// TIA Portal V21 export
FUNCTION "PassiLavaggio_010102" : Void   // FC102, LAD
{ S7_Optimized_Access := 'TRUE' }
// stored: SetENOAutomatically false
   VAR_TEMP
      CondizioniPassoEsterne : Bool;
      AbilitazionePasso : Bool;
      AppoggioComando : Int;
      ComandoValvolaG : Int;
      ComandoValvolaA1 : Int;
      PompaPistoniAbilitata : Bool;
   END_VAR
   VAR CONSTANT
      Positivo : Int := 2;
      Negativo : Int := 3;
      FolleScarico : Int := 4;
      FlipFlop : Int := 5;
   END_VAR
BEGIN

REGION Network 1: Sequenza: Lavaggio - Passo: Risciacquo. Condizioni passo esterne.
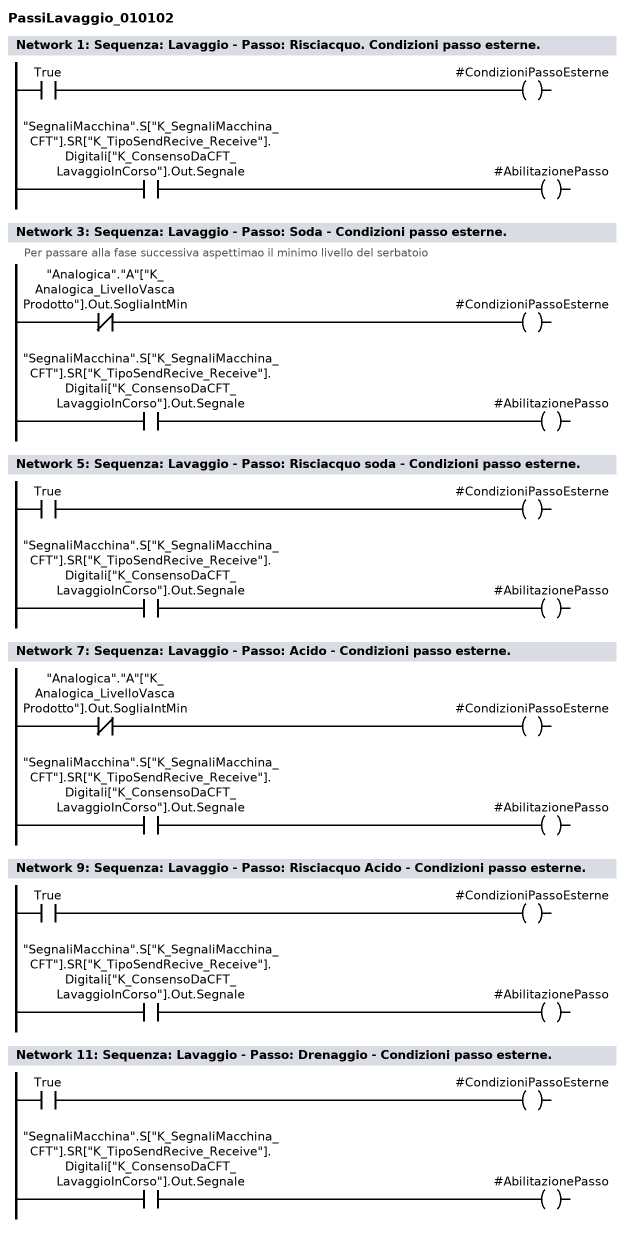
   RUNG wire#powerrail
      Contact( True )
      Coil( #CondizioniPassoEsterne )
   END_RUNG
   RUNG wire#powerrail
      Contact( "SegnaliMacchina".S["K_SegnaliMacchina_CFT"].SR["K_TipoSendRecive_Receive"].Digitali["K_ConsensoDaCFT_LavaggioInCorso"].Out.Segnale )
      Coil( #AbilitazionePasso )
   END_RUNG
   // the same network as SCL:
   #CondizioniPassoEsterne := True;
   #AbilitazionePasso := "SegnaliMacchina".S["K_SegnaliMacchina_CFT"].SR["K_TipoSendRecive_Receive"].Digitali["K_ConsensoDaCFT_LavaggioInCorso"].Out.Segnale;
END_REGION

REGION Network 2 (SCL): Sequenza: Lavaggio - Passo: Risciacquo. Gestione del passo.
   REGION Parametri del passo
       "GestPasso"(K_PassoAttuale := "K_Passo_Risciacquo",
                   K_PassoSuccessivo := "K_Passo_Soda",
                   AbilitaSaltapasso := True,
                   AbilitaPasso:= #AbilitazionePasso,
                   CondizioniPassoEsterne := #CondizioniPassoEsterne,
                   K_Sequenza := "K_Sequenza_Lavaggio");
   END_REGION ;
   REGION Comando delle utenze nel passo

       "GestPasso_CmdValvola"(K_Valvola := "K_Valvola_A1",
                              Comando := #Positivo,
                              K_Sequenza := "K_Sequenza_Lavaggio",
                              K_Passo := "K_Passo_Risciacquo",
                              NonAttenderePosizione:= "Analogica".A[K_Analogica_LivelloVascaProdotto].Out.SogliaIntMax);

       "GestPasso_CmdValvola"(K_Valvola := "K_Valvola_A",
                              Comando := #Positivo,
                              K_Sequenza := "K_Sequenza_Lavaggio",
                              K_Passo := "K_Passo_Risciacquo",
                              NonAttenderePosizione := "Analogica".A[K_Analogica_LivelloVascaProdotto].Out.SogliaIntMax);

       "GestPasso_CmdValvolaFlipFlop"(K_Valvola := "K_Valvola_B",
                                      NumeroCicli := 3,
                                      TempoPositivo := "Sequenza".S[K_Sequenza_Lavaggio].Prm.Passo[K_Passo_Risciacquo].Durata.Preset / 3,  //Tempo a ricetta per immissione soda
                                      TempoNegativo := 5,
                                      ComandoARiposo:=#Positivo,
                                      K_Sequenza := "K_Sequenza_Lavaggio",
                                      K_Passo := "K_Passo_Risciacquo");

       "GestPasso_CmdValvola"(K_Valvola := "K_Valvola_B1",
                              Comando := "GestPasso_ReplicaComandoValvola"("K_Valvola_B"),
                              K_Sequenza := "K_Sequenza_Lavaggio",
                              K_Passo := "K_Passo_Risciacquo",
                              NonAttenderePosizione:= False);

       "GestPasso_CmdValvola"(K_Valvola := "K_Valvola_E",
                              Comando := #Positivo,
                              K_Sequenza := "K_Sequenza_Lavaggio",
                              K_Passo := "K_Passo_Risciacquo",
                              NonAttenderePosizione:= False);

       "GestPasso_CmdValvola"(K_Valvola := "K_Valvola_E1",
                              Comando := #Positivo,
                              K_Sequenza := "K_Sequenza_Lavaggio",
                              K_Passo := "K_Passo_Risciacquo",
                              NonAttenderePosizione:= False);

       "GestPasso_CmdValvola"(K_Valvola := "K_Valvola_G",
                              Comando := #Positivo,
                              K_Sequenza := "K_Sequenza_Lavaggio",
                              K_Passo := "K_Passo_Risciacquo",
                              NonAttenderePosizione := False);

       "GestPasso_CmdValvolaFlipFlop"(K_Valvola := "K_Valvola_CP1",
                                      NumeroCicli := 5,
                                      TempoPositivo := "Sequenza".S[K_Sequenza_Lavaggio].Prm.Passo[K_Passo_Risciacquo].Durata.Preset / 5,
                                      TempoNegativo := 5,
                                      ComandoARiposo:=#Positivo,
                                      K_Passo := "K_Passo_Risciacquo",
                                      K_Sequenza := "K_Sequenza_Lavaggio");

       "GestPasso_CmdMotore"(K_Motore := "K_Motore_PompaMono",
                             Comando := #Positivo,
                             K_Sequenza := "K_Sequenza_Lavaggio",
                             K_Passo := "K_Passo_Risciacquo",
                             NonAttenderePosizione := False);
       #PompaPistoniAbilitata := "MacchinaARicetta".M[K_MacchinaARicetta_SterilizzatoreTubo].Lavoro.DatoBool[K_DatoRicettaBool_SterilizzatoreTubo_AbilitazionePompaPistoni];
       IF #PompaPistoniAbilitata THEN
           "GestPasso_CmdMotore"(K_Motore := "K_Motore_PompaPistoni",
                                 Comando := #Positivo,
                                 K_Sequenza := "K_Sequenza_Lavaggio",
                                 K_Passo := "K_Passo_Risciacquo",
                                 NonAttenderePosizione := NOT "MacchinaARicetta".M[K_MacchinaARicetta_SterilizzatoreTubo].Lavoro.DatoBool[K_DatoRicettaBool_SterilizzatoreTubo_AbilitazionePompaPistoni]);
       END_IF;
       "GestPasso_CmdMotore"(K_Motore := "K_Motore_CentrifugaLavaggio",
                             Comando := #Positivo,
                             K_Sequenza := "K_Sequenza_Lavaggio",
                             K_Passo := "K_Passo_Risciacquo",
                             NonAttenderePosizione := False);
   END_REGION ;
END_REGION

REGION Network 3: Sequenza: Lavaggio - Passo: Soda - Condizioni passo esterne.
   // Per passare alla fase successiva aspettimao il minimo livello del serbatoio
   RUNG wire#powerrail
      I_Contact( "Analogica"."A"["K_Analogica_LivelloVascaProdotto"].Out.SogliaIntMin )
      Coil( #CondizioniPassoEsterne )
   END_RUNG
   RUNG wire#powerrail
      Contact( "SegnaliMacchina".S["K_SegnaliMacchina_CFT"].SR["K_TipoSendRecive_Receive"].Digitali["K_ConsensoDaCFT_LavaggioInCorso"].Out.Segnale )
      Coil( #AbilitazionePasso )
   END_RUNG
   // the same network as SCL:
   #CondizioniPassoEsterne := NOT "Analogica"."A"["K_Analogica_LivelloVascaProdotto"].Out.SogliaIntMin;
   #AbilitazionePasso := "SegnaliMacchina".S["K_SegnaliMacchina_CFT"].SR["K_TipoSendRecive_Receive"].Digitali["K_ConsensoDaCFT_LavaggioInCorso"].Out.Segnale;
END_REGION

REGION Network 4 (SCL): Sequenza: Lavaggio - Passo: Soda - Gestione del passo.
   REGION Parametri del passo
       "GestPasso"(K_PassoAttuale := "K_Passo_Soda",
                   K_PassoSuccessivo := "K_Passo_RisciacquoSoda",
                   AbilitaSaltapasso := True,
                   AbilitaPasso:= #AbilitazionePasso,
                   CondizioniPassoEsterne := #CondizioniPassoEsterne,
                   K_Sequenza := "K_Sequenza_Lavaggio");
   END_REGION ;
   REGION Comando delle utenze nel passo    
       IF "Sequenza".S[K_Sequenza_Lavaggio].Prm.Passo[K_Passo_Soda].Durata.O THEN
           #ComandoValvolaA1 := #Negativo;
       ELSE
           #ComandoValvolaA1 := #Positivo;
       END_IF;
       "GestPasso_CmdValvola"(K_Valvola := "K_Valvola_A1",
                              Comando := #ComandoValvolaA1,
                              K_Sequenza := "K_Sequenza_Lavaggio",
                              K_Passo := "K_Passo_Soda",
                              NonAttenderePosizione:= "Analogica".A[K_Analogica_LivelloVascaProdotto].Out.SogliaIntMax);

       "GestPasso_CmdValvola"(K_Valvola := "K_Valvola_A",
                              Comando := #ComandoValvolaA1,
                              K_Sequenza := "K_Sequenza_Lavaggio",
                              K_Passo := "K_Passo_Soda",
                              NonAttenderePosizione := "Analogica".A[K_Analogica_LivelloVascaProdotto].Out.SogliaIntMax);

       "GestPasso_CmdValvolaFlipFlop"(K_Valvola := "K_Valvola_B",
                                      NumeroCicli := 8,
                                      TempoPositivo := "Sequenza".S[K_Sequenza_Lavaggio].Prm.Passo[K_Passo_Soda].Durata.Preset / 8,
                                      TempoNegativo := 5,
                                      ComandoARiposo:=#Positivo,
                                      K_Passo := "K_Passo_Soda",
                                      K_Sequenza := "K_Sequenza_Lavaggio");

       "GestPasso_CmdValvola"(K_Valvola := "K_Valvola_B1",
                              Comando := "GestPasso_ReplicaComandoValvola"("K_Valvola_B"),
                              K_Sequenza := "K_Sequenza_Lavaggio",
                              K_Passo := "K_Passo_Soda",
                              NonAttenderePosizione:= False);

       "GestPasso_CmdValvola"(K_Valvola := "K_Valvola_D",
                              Comando := #Positivo,
                              K_Sequenza := "K_Sequenza_Lavaggio",
                              K_Passo := "K_Passo_Soda",
                              NonAttenderePosizione:= False);

       "GestPasso_CmdValvola"(K_Valvola := "K_Valvola_D2",
                              Comando :=#Positivo,
                              K_Sequenza := "K_Sequenza_Lavaggio",
                              K_Passo := "K_Passo_Soda",
                              NonAttenderePosizione:= False);

       "GestPasso_CmdValvola"(K_Valvola := "K_Valvola_E",
                              Comando := #Positivo,
                              K_Sequenza := "K_Sequenza_Lavaggio",
                              K_Passo := "K_Passo_Soda",
                              NonAttenderePosizione:= False);

       "GestPasso_CmdValvola"(K_Valvola := "K_Valvola_E1",
                              Comando := #Positivo,
                              K_Sequenza := "K_Sequenza_Lavaggio",
                              K_Passo := "K_Passo_Soda",
                              NonAttenderePosizione:= False);

       REGION Valvola G
           //Al termine del passo prima di passare al passo successivo aspetto il livello minimo,
           //quindi metto in scarico invece di andare in vasca.
           IF "Sequenza".S[K_Sequenza_Lavaggio].Prm.Passo[K_Passo_Soda].Durata.O THEN
               #ComandoValvolaG := #Positivo;
           ELSE
               #ComandoValvolaG := #Negativo;
           END_IF;

           "GestPasso_CmdValvola"(K_Valvola := "K_Valvola_G",
                                  Comando := #ComandoValvolaG,
                                  K_Sequenza := "K_Sequenza_Lavaggio",
                                  K_Passo := "K_Passo_Soda",
                                  NonAttenderePosizione := False);
       END_REGION ;

       "GestPasso_CmdValvola"(K_Valvola := "K_Valvola_Z1",
                              Comando := "GestPasso_ReplicaComandoValvola"("K_Valvola_XXX"),
                              K_Sequenza := "K_Sequenza_Lavaggio",
                              K_Passo := "K_Passo_Soda",
                              NonAttenderePosizione:= False);

       "GestPasso_CmdValvolaFlipFlop"(K_Valvola := "K_Valvola_XXX",
                                      NumeroCicli := 1,
                                      TempoPositivo := 300,  //Tempo per immissione soda
                                      TempoNegativo := 0,
                                      ComandoARiposo:=#Negativo,
                                      K_Sequenza := "K_Sequenza_Lavaggio",
                                      K_Passo := "K_Passo_Soda");

       "GestPasso_CmdValvolaFlipFlop"(K_Valvola := "K_Valvola_CP1",
                                      NumeroCicli := 5,
                                      TempoPositivo := "Sequenza".S[K_Sequenza_Lavaggio].Prm.Passo[K_Passo_Soda].Durata.Preset / 5,
                                      TempoNegativo := 5,
                                      ComandoARiposo:=#Positivo,
                                      K_Passo := "K_Passo_Soda",
                                      K_Sequenza := "K_Sequenza_Lavaggio");
       //Motori
       "GestPasso_CmdMotore"(K_Motore := "K_Motore_PompaMono",
                             Comando := #Positivo,
                             K_Sequenza := "K_Sequenza_Lavaggio",
                             K_Passo := "K_Passo_Soda",
                             NonAttenderePosizione := False);
       IF #PompaPistoniAbilitata THEN
           "GestPasso_CmdMotore"(K_Motore := "K_Motore_PompaPistoni",
                                 Comando := #Positivo,
                                 K_Sequenza := "K_Sequenza_Lavaggio",
                                 K_Passo := "K_Passo_Soda",
                                 NonAttenderePosizione := NOT "MacchinaARicetta".M[K_MacchinaARicetta_SterilizzatoreTubo].Lavoro.DatoBool[K_DatoRicettaBool_SterilizzatoreTubo_AbilitazionePompaPistoni]);
       END_IF;
       "GestPasso_CmdMotore"(K_Motore := "K_Motore_CentrifugaLavaggio",
                             Comando := #Positivo,
                             K_Sequenza := "K_Sequenza_Lavaggio",
                             K_Passo := "K_Passo_Soda",
                             NonAttenderePosizione := False);

       "GestPasso_CmdMotore"(K_Motore := "K_Motore_PompaRicircoloAcquaCalda",
                             Comando := #Positivo,
                             K_Sequenza := "K_Sequenza_Lavaggio",
                             K_Passo := "K_Passo_Soda",
                             NonAttenderePosizione := False);

   END_REGION ;
END_REGION

REGION Network 5: Sequenza: Lavaggio - Passo: Risciacquo soda - Condizioni passo esterne.
   RUNG wire#powerrail
      Contact( True )
      Coil( #CondizioniPassoEsterne )
   END_RUNG
   RUNG wire#powerrail
      Contact( "SegnaliMacchina".S["K_SegnaliMacchina_CFT"].SR["K_TipoSendRecive_Receive"].Digitali["K_ConsensoDaCFT_LavaggioInCorso"].Out.Segnale )
      Coil( #AbilitazionePasso )
   END_RUNG
   // the same network as SCL:
   #CondizioniPassoEsterne := True;
   #AbilitazionePasso := "SegnaliMacchina".S["K_SegnaliMacchina_CFT"].SR["K_TipoSendRecive_Receive"].Digitali["K_ConsensoDaCFT_LavaggioInCorso"].Out.Segnale;
END_REGION

REGION Network 6 (SCL): Sequenza: Lavaggio - Passo: Risciacquo soda - Gestione del passo.
   REGION Parametri del passo
   "GestPasso"(K_PassoAttuale := "K_Passo_RisciacquoSoda",
               K_PassoSuccessivo := "K_Passo_Acido",
               AbilitaSaltapasso := True,
               AbilitaPasso:= #AbilitazionePasso,
               CondizioniPassoEsterne := #CondizioniPassoEsterne,
               K_Sequenza := "K_Sequenza_Lavaggio");
   END_REGION ;
   REGION Comando delle utenze nel passo
       "GestPasso_CmdValvola"(K_Valvola := "K_Valvola_A1",
                              Comando := #Positivo,
                              K_Sequenza := "K_Sequenza_Lavaggio",
                              K_Passo := "K_Passo_RisciacquoSoda",
                              NonAttenderePosizione := "Analogica".A[K_Analogica_LivelloVascaProdotto].Out.SogliaIntMax);

       "GestPasso_CmdValvola"(K_Valvola := "K_Valvola_A",
                              Comando := #Positivo,
                              K_Sequenza := "K_Sequenza_Lavaggio",
                              K_Passo := "K_Passo_RisciacquoSoda",
                              NonAttenderePosizione := "Analogica".A[K_Analogica_LivelloVascaProdotto].Out.SogliaIntMax);

       "GestPasso_CmdValvolaFlipFlop"(K_Valvola := "K_Valvola_B",
                                      NumeroCicli := 3,
                                      TempoPositivo := "Sequenza".S[K_Sequenza_Lavaggio].Prm.Passo[K_Passo_RisciacquoSoda].Durata.Preset / 3,  //Tempo a ricetta per immissione soda
                                      TempoNegativo := 5,
                                      ComandoARiposo:=#Positivo,
                                      K_Sequenza := "K_Sequenza_Lavaggio",
                                      K_Passo := "K_Passo_RisciacquoSoda");

       "GestPasso_CmdValvola"(K_Valvola := "K_Valvola_B1",
                              Comando := "GestPasso_ReplicaComandoValvola"("K_Valvola_B"),
                              K_Sequenza := "K_Sequenza_Lavaggio",
                              K_Passo := "K_Passo_RisciacquoSoda",
                              NonAttenderePosizione := False);

       "GestPasso_CmdValvola"(K_Valvola := "K_Valvola_E",
                              Comando := #Positivo,
                              K_Sequenza := "K_Sequenza_Lavaggio",
                              K_Passo := "K_Passo_RisciacquoSoda",
                              NonAttenderePosizione := False);

       "GestPasso_CmdValvola"(K_Valvola := "K_Valvola_E1",
                              Comando := #Positivo,
                              K_Sequenza := "K_Sequenza_Lavaggio",
                              K_Passo := "K_Passo_RisciacquoSoda",
                              NonAttenderePosizione := False);

       "GestPasso_CmdValvola"(K_Valvola := "K_Valvola_G",
                              Comando := #Positivo,
                              K_Sequenza := "K_Sequenza_Lavaggio",
                              K_Passo := "K_Passo_RisciacquoSoda",
                              NonAttenderePosizione := False);

       "GestPasso_CmdValvolaFlipFlop"(K_Valvola := "K_Valvola_CP1",
                                      NumeroCicli := 5,
                                      TempoPositivo := "Sequenza".S[K_Sequenza_Lavaggio].Prm.Passo[K_Passo_RisciacquoSoda].Durata.Preset / 5,
                                      TempoNegativo := 5,
                                      ComandoARiposo:=#Positivo,
                                      K_Passo := "K_Passo_RisciacquoSoda",
                                      K_Sequenza := "K_Sequenza_Lavaggio");

       "GestPasso_CmdMotore"(K_Motore := "K_Motore_PompaMono",
                             Comando := #Positivo,
                             K_Sequenza := "K_Sequenza_Lavaggio",
                             K_Passo := "K_Passo_RisciacquoSoda",
                             NonAttenderePosizione := False);
       IF #PompaPistoniAbilitata THEN
           "GestPasso_CmdMotore"(K_Motore := "K_Motore_PompaPistoni",
                                 Comando := #Positivo,
                                 K_Sequenza := "K_Sequenza_Lavaggio",
                                 K_Passo := "K_Passo_RisciacquoSoda",
                                 NonAttenderePosizione := NOT "MacchinaARicetta".M[K_MacchinaARicetta_SterilizzatoreTubo].Lavoro.DatoBool[K_DatoRicettaBool_SterilizzatoreTubo_AbilitazionePompaPistoni]);
       END_IF;
       "GestPasso_CmdMotore"(K_Motore := "K_Motore_CentrifugaLavaggio",
                             Comando := #Positivo,
                             K_Sequenza := "K_Sequenza_Lavaggio",
                             K_Passo := "K_Passo_RisciacquoSoda",
                             NonAttenderePosizione := False);
   END_REGION ;
END_REGION

REGION Network 7: Sequenza: Lavaggio - Passo: Acido - Condizioni passo esterne.
   RUNG wire#powerrail
      I_Contact( "Analogica"."A"["K_Analogica_LivelloVascaProdotto"].Out.SogliaIntMin )
      Coil( #CondizioniPassoEsterne )
   END_RUNG
   RUNG wire#powerrail
      Contact( "SegnaliMacchina".S["K_SegnaliMacchina_CFT"].SR["K_TipoSendRecive_Receive"].Digitali["K_ConsensoDaCFT_LavaggioInCorso"].Out.Segnale )
      Coil( #AbilitazionePasso )
   END_RUNG
   // the same network as SCL:
   #CondizioniPassoEsterne := NOT "Analogica"."A"["K_Analogica_LivelloVascaProdotto"].Out.SogliaIntMin;
   #AbilitazionePasso := "SegnaliMacchina".S["K_SegnaliMacchina_CFT"].SR["K_TipoSendRecive_Receive"].Digitali["K_ConsensoDaCFT_LavaggioInCorso"].Out.Segnale;
END_REGION

REGION Network 8 (SCL): Sequenza: Lavaggio - Passo: Acido - Gestione del passo.
   REGION Parametri del passo
       "GestPasso"(K_PassoAttuale := "K_Passo_Acido",
                   K_PassoSuccessivo := "K_Passo_RisciacquoAcido",
                   AbilitaSaltapasso := True,
                   AbilitaPasso:= #AbilitazionePasso,
                   CondizioniPassoEsterne := #CondizioniPassoEsterne,
                   K_Sequenza := "K_Sequenza_Lavaggio");
   END_REGION ;
   REGION Comando delle utenze nel passo    
       IF "Sequenza".S[K_Sequenza_Lavaggio].Prm.Passo[K_Passo_Acido].Durata.O THEN
           #ComandoValvolaA1 := #Negativo;
       ELSE
           #ComandoValvolaA1 := #Positivo;
       END_IF;
       "GestPasso_CmdValvola"(K_Valvola := "K_Valvola_A1",
                              Comando := #ComandoValvolaA1,
                              K_Sequenza := "K_Sequenza_Lavaggio",
                              K_Passo := "K_Passo_Acido",
                              NonAttenderePosizione := "Analogica".A[K_Analogica_LivelloVascaProdotto].Out.SogliaIntMax);

       "GestPasso_CmdValvola"(K_Valvola := "K_Valvola_A",
                              Comando := #ComandoValvolaA1,
                              K_Sequenza := "K_Sequenza_Lavaggio",
                              K_Passo := "K_Passo_Acido",
                              NonAttenderePosizione := "Analogica".A[K_Analogica_LivelloVascaProdotto].Out.SogliaIntMax);

       "GestPasso_CmdValvolaFlipFlop"(K_Valvola := "K_Valvola_B",
                                      NumeroCicli := 8,
                                      TempoPositivo := "Sequenza".S[K_Sequenza_Lavaggio].Prm.Passo[K_Passo_Acido].Durata.Preset / 8,
                                      TempoNegativo := 5,
                                      ComandoARiposo:=#Positivo,
                                      K_Passo := "K_Passo_Acido",
                                      K_Sequenza := "K_Sequenza_Lavaggio");

       "GestPasso_CmdValvola"(K_Valvola := "K_Valvola_B1",
                              Comando := "GestPasso_ReplicaComandoValvola"("K_Valvola_B"),
                              K_Sequenza := "K_Sequenza_Lavaggio",
                              K_Passo := "K_Passo_Acido",
                              NonAttenderePosizione := False);

       "GestPasso_CmdValvola"(K_Valvola := "K_Valvola_D",
                              Comando := #Positivo,
                              K_Sequenza := "K_Sequenza_Lavaggio",
                              K_Passo := "K_Passo_Acido",
                              NonAttenderePosizione := False);

       "GestPasso_CmdValvola"(K_Valvola := "K_Valvola_D2",
                              Comando := #Positivo,
                              K_Sequenza := "K_Sequenza_Lavaggio",
                              K_Passo := "K_Passo_Acido",
                              NonAttenderePosizione := False);

       "GestPasso_CmdValvola"(K_Valvola := "K_Valvola_E",
                              Comando := #Positivo,
                              K_Sequenza := "K_Sequenza_Lavaggio",
                              K_Passo := "K_Passo_Acido",
                              NonAttenderePosizione := False);

       "GestPasso_CmdValvola"(K_Valvola := "K_Valvola_E1",
                              Comando := #Positivo,
                              K_Sequenza := "K_Sequenza_Lavaggio",
                              K_Passo := "K_Passo_Acido",
                              NonAttenderePosizione := False);

       "GestPasso_CmdValvola"(K_Valvola := "K_Valvola_Y",
                              Comando := #Positivo,
                              K_Sequenza := "K_Sequenza_Lavaggio",
                              K_Passo := "K_Passo_Acido",
                              NonAttenderePosizione := False);

       "GestPasso_CmdValvola"(K_Valvola := "K_Valvola_Y1",
                              Comando := #Positivo,
                              K_Sequenza := "K_Sequenza_Lavaggio",
                              K_Passo := "K_Passo_Acido",
                              NonAttenderePosizione := False);
       REGION Valvola G
           //Al termine del passo prima di passare al passo successivo aspetto il livello minimo,
           //quindi metto in scarico invece di andare in vasca.
           IF "Sequenza".S[K_Sequenza_Lavaggio].Prm.Passo[K_Passo_Acido].Durata.O THEN
               #ComandoValvolaG := #Positivo;
           ELSE
               #ComandoValvolaG := #Negativo;
           END_IF;

           "GestPasso_CmdValvola"(K_Valvola := "K_Valvola_G",
                                  Comando := #ComandoValvolaG,
                                  K_Sequenza := "K_Sequenza_Lavaggio",
                                  K_Passo := "K_Passo_Acido",
                                  NonAttenderePosizione := False);
       END_REGION ;

       "GestPasso_CmdValvola"(K_Valvola := "K_Valvola_Z1",
                              Comando := "GestPasso_ReplicaComandoValvola"("K_Valvola_XX"),
                              K_Sequenza := "K_Sequenza_Lavaggio",
                              K_Passo := "K_Passo_Acido",
                              NonAttenderePosizione := False);

       "GestPasso_CmdValvolaFlipFlop"(K_Valvola := "K_Valvola_XX",
                                      NumeroCicli := 1,
                                      TempoPositivo := 300,  //Tempo per immissione acido
                                      TempoNegativo := 0,
                                      ComandoARiposo:=#Negativo,
                                      K_Sequenza := "K_Sequenza_Lavaggio",
                                      K_Passo := "K_Passo_Acido");

       "GestPasso_CmdValvolaFlipFlop"(K_Valvola := "K_Valvola_CP1",
                                      NumeroCicli := 5,
                                      TempoPositivo := "Sequenza".S[K_Sequenza_Lavaggio].Prm.Passo[K_Passo_Acido].Durata.Preset / 5,
                                      TempoNegativo := 5,
                                      ComandoARiposo:=#Positivo,
                                      K_Passo := "K_Passo_Acido",
                                      K_Sequenza := "K_Sequenza_Lavaggio");
       //Motori
       "GestPasso_CmdMotore"(K_Motore := "K_Motore_PompaMono",
                             Comando := #Positivo,
                             K_Sequenza := "K_Sequenza_Lavaggio",
                             K_Passo := "K_Passo_Acido",
                             NonAttenderePosizione := False);
       IF #PompaPistoniAbilitata THEN
           "GestPasso_CmdMotore"(K_Motore := "K_Motore_PompaPistoni",
                                 Comando := #Positivo,
                                 K_Sequenza := "K_Sequenza_Lavaggio",
                                 K_Passo := "K_Passo_Acido",
                                 NonAttenderePosizione := NOT "MacchinaARicetta".M[K_MacchinaARicetta_SterilizzatoreTubo].Lavoro.DatoBool[K_DatoRicettaBool_SterilizzatoreTubo_AbilitazionePompaPistoni]);
       END_IF;
       "GestPasso_CmdMotore"(K_Motore := "K_Motore_CentrifugaLavaggio",
                             Comando := #Positivo,
                             K_Sequenza := "K_Sequenza_Lavaggio",
                             K_Passo := "K_Passo_Acido",
                             NonAttenderePosizione := False);

       "GestPasso_CmdMotore"(K_Motore := "K_Motore_PompaRicircoloAcquaCalda",
                             Comando := #Positivo,
                             K_Sequenza := "K_Sequenza_Lavaggio",
                             K_Passo := "K_Passo_Acido",
                             NonAttenderePosizione := False);
   END_REGION ;
END_REGION

REGION Network 9: Sequenza: Lavaggio - Passo: Risciacquo Acido - Condizioni passo esterne.
   RUNG wire#powerrail
      Contact( True )
      Coil( #CondizioniPassoEsterne )
   END_RUNG
   RUNG wire#powerrail
      Contact( "SegnaliMacchina".S["K_SegnaliMacchina_CFT"].SR["K_TipoSendRecive_Receive"].Digitali["K_ConsensoDaCFT_LavaggioInCorso"].Out.Segnale )
      Coil( #AbilitazionePasso )
   END_RUNG
   // the same network as SCL:
   #CondizioniPassoEsterne := True;
   #AbilitazionePasso := "SegnaliMacchina".S["K_SegnaliMacchina_CFT"].SR["K_TipoSendRecive_Receive"].Digitali["K_ConsensoDaCFT_LavaggioInCorso"].Out.Segnale;
END_REGION

REGION Network 10 (SCL): Sequenza: Lavaggio - Passo: Risciacquo Acido - Gestione del passo.
   REGION Parametri del passo
       "GestPasso"(K_PassoAttuale := "K_Passo_RisciacquoAcido",
                   K_PassoSuccessivo := "K_Passo_Drenaggio",
                   AbilitaSaltapasso := True,
                   AbilitaPasso:= #AbilitazionePasso,
                   CondizioniPassoEsterne := #CondizioniPassoEsterne,
                   K_Sequenza := "K_Sequenza_Lavaggio");
   END_REGION ;
   REGION Comando delle utenze nel passo    
       "GestPasso_CmdValvola"(K_Valvola := "K_Valvola_A1",
                              Comando := #Positivo,
                              K_Sequenza := "K_Sequenza_Lavaggio",
                              K_Passo := "K_Passo_RisciacquoAcido",
                              NonAttenderePosizione := "Analogica".A[K_Analogica_LivelloVascaProdotto].Out.SogliaIntMax);

       "GestPasso_CmdValvola"(K_Valvola := "K_Valvola_A",
                              Comando := #Positivo,
                              K_Sequenza := "K_Sequenza_Lavaggio",
                              K_Passo := "K_Passo_RisciacquoAcido",
                              NonAttenderePosizione := "Analogica".A[K_Analogica_LivelloVascaProdotto].Out.SogliaIntMax);

       "GestPasso_CmdValvolaFlipFlop"(K_Valvola := "K_Valvola_B",
                                      NumeroCicli := 3,
                                      TempoPositivo := "Sequenza".S[K_Sequenza_Lavaggio].Prm.Passo[K_Passo_RisciacquoAcido].Durata.Preset / 3,  //Tempo a ricetta per immissione soda
                                      TempoNegativo := 5,
                                      ComandoARiposo:=#Positivo,
                                      K_Sequenza := "K_Sequenza_Lavaggio",
                                      K_Passo := "K_Passo_RisciacquoAcido");

       "GestPasso_CmdValvola"(K_Valvola := "K_Valvola_B1",
                              Comando := "GestPasso_ReplicaComandoValvola"("K_Valvola_B"),
                              K_Sequenza := "K_Sequenza_Lavaggio",
                              K_Passo := "K_Passo_RisciacquoAcido",
                              NonAttenderePosizione := False);

       "GestPasso_CmdValvola"(K_Valvola := "K_Valvola_E",
                              Comando := #Positivo,
                              K_Sequenza := "K_Sequenza_Lavaggio",
                              K_Passo := "K_Passo_RisciacquoAcido",
                              NonAttenderePosizione := False);

       "GestPasso_CmdValvola"(K_Valvola := "K_Valvola_E1",
                              Comando := #Positivo,
                              K_Sequenza := "K_Sequenza_Lavaggio",
                              K_Passo := "K_Passo_RisciacquoAcido",
                              NonAttenderePosizione := False);

       "GestPasso_CmdValvola"(K_Valvola := "K_Valvola_G",
                              Comando := #Positivo,
                              K_Sequenza := "K_Sequenza_Lavaggio",
                              K_Passo := "K_Passo_RisciacquoAcido",
                              NonAttenderePosizione := False);

       "GestPasso_CmdValvola"(K_Valvola := "K_Valvola_Y",
                              Comando := #Positivo,
                              K_Sequenza := "K_Sequenza_Lavaggio",
                              K_Passo := "K_Passo_RisciacquoAcido",
                              NonAttenderePosizione := False);

       "GestPasso_CmdValvola"(K_Valvola := "K_Valvola_Y1",
                              Comando := #Positivo,
                              K_Sequenza := "K_Sequenza_Lavaggio",
                              K_Passo := "K_Passo_RisciacquoAcido",
                              NonAttenderePosizione := False);

       "GestPasso_CmdValvolaFlipFlop"(K_Valvola := "K_Valvola_CP1",
                                      NumeroCicli := 5,
                                      TempoPositivo := "Sequenza".S[K_Sequenza_Lavaggio].Prm.Passo[K_Passo_RisciacquoAcido].Durata.Preset / 5,
                                      TempoNegativo := 5,
                                      ComandoARiposo:=#Positivo,
                                      K_Passo := "K_Passo_RisciacquoAcido",
                                      K_Sequenza := "K_Sequenza_Lavaggio");

       "GestPasso_CmdMotore"(K_Motore := "K_Motore_PompaMono",
                             Comando := #Positivo,
                             K_Sequenza := "K_Sequenza_Lavaggio",
                             K_Passo := "K_Passo_RisciacquoAcido",
                             NonAttenderePosizione := False);
       IF #PompaPistoniAbilitata THEN
           "GestPasso_CmdMotore"(K_Motore := "K_Motore_PompaPistoni",
                                 Comando := #Positivo,
                                 K_Sequenza := "K_Sequenza_Lavaggio",
                                 K_Passo := "K_Passo_RisciacquoAcido",
                                 NonAttenderePosizione := NOT "MacchinaARicetta".M[K_MacchinaARicetta_SterilizzatoreTubo].Lavoro.DatoBool[K_DatoRicettaBool_SterilizzatoreTubo_AbilitazionePompaPistoni]);
       END_IF;
       "GestPasso_CmdMotore"(K_Motore := "K_Motore_CentrifugaLavaggio",
                             Comando := #Positivo,
                             K_Sequenza := "K_Sequenza_Lavaggio",
                             K_Passo := "K_Passo_RisciacquoAcido",
                             NonAttenderePosizione := False);
   END_REGION ;
END_REGION

REGION Network 11: Sequenza: Lavaggio - Passo: Drenaggio - Condizioni passo esterne.
   RUNG wire#powerrail
      Contact( True )
      Coil( #CondizioniPassoEsterne )
   END_RUNG
   RUNG wire#powerrail
      Contact( "SegnaliMacchina".S["K_SegnaliMacchina_CFT"].SR["K_TipoSendRecive_Receive"].Digitali["K_ConsensoDaCFT_LavaggioInCorso"].Out.Segnale )
      Coil( #AbilitazionePasso )
   END_RUNG
   // the same network as SCL:
   #CondizioniPassoEsterne := True;
   #AbilitazionePasso := "SegnaliMacchina".S["K_SegnaliMacchina_CFT"].SR["K_TipoSendRecive_Receive"].Digitali["K_ConsensoDaCFT_LavaggioInCorso"].Out.Segnale;
END_REGION

REGION Network 12 (SCL): Sequenza: Lavaggio - Passo: Drenaggio - Gestione del passo.
   REGION Parametri del passo
       "GestPasso"(K_PassoAttuale := "K_Passo_Drenaggio",
                   K_PassoSuccessivo := 0,
                   AbilitaSaltapasso := True,
                   AbilitaPasso:= #AbilitazionePasso,
                   CondizioniPassoEsterne := #CondizioniPassoEsterne,
                   K_Sequenza := "K_Sequenza_Lavaggio");
   END_REGION ;
   REGION Comando delle utenze nel passo    
       "GestPasso_CmdValvola"(K_Valvola := "K_Valvola_B",
                              Comando := #Positivo,
                              K_Sequenza := "K_Sequenza_Lavaggio",
                              K_Passo := "K_Passo_Drenaggio",
                              NonAttenderePosizione:= False);

       "GestPasso_CmdValvola"(K_Valvola := "K_Valvola_B1",
                              Comando := "GestPasso_ReplicaComandoValvola"("K_Valvola_B"),
                              K_Sequenza := "K_Sequenza_Lavaggio",
                              K_Passo := "K_Passo_Drenaggio",
                              NonAttenderePosizione:= False);

       "GestPasso_CmdValvola"(K_Valvola := "K_Valvola_C",
                              Comando := #Positivo,
                              K_Sequenza := "K_Sequenza_Lavaggio",
                              K_Passo := "K_Passo_Drenaggio",
                              NonAttenderePosizione:= False);

       "GestPasso_CmdValvola"(K_Valvola := "K_Valvola_H",
                              Comando := #Positivo,
                              K_Sequenza := "K_Sequenza_Lavaggio",
                              K_Passo := "K_Passo_Drenaggio",
                              NonAttenderePosizione:= False);

       "GestPasso_CmdValvola"(K_Valvola := "K_Valvola_H1",
                              Comando := #Positivo,
                              K_Sequenza := "K_Sequenza_Lavaggio",
                              K_Passo := "K_Passo_Drenaggio",
                              NonAttenderePosizione:= False);
   END_REGION ;
END_REGION
END_FUNCTION
